(* PLC project Pizzarpocessor_03_11_2025.project, CODESYS CODESYS V3.5 SP21 Patch 1 *)
(* stored: creationDateTime 2025-11-18T11:47:58.0390156, modificationDateTime 2025-11-12T10:55:39.9225124 *)

TYPE HopperState : (OFF, IDLE, DISPENSING, LOW_LEVEL_FAULT, BLOCKED, MANUAL);
END_TYPE

TYPE ConveyorStatus : STRUCT
  Conveyor_ID : INT;  (* Conveyor number/ID *)
  Speed : REAL;  (* Percentage of speed *)
  Running : BOOL;
  State : ConveyorState;
  Ready : BOOL;  (* Interlock *)
END_STRUCT;
END_TYPE

TYPE HopperStatus : STRUCT
  Hopper_Id : INT;  (* Hopper Location/ID *)
  State : HopperState;  (* HopperState refering to ENUM *)
  Fill_Level : REAL;  (* Hopper_Ingredient level *)
  Ingredient_ID : INT;  (* Ingredient Name or Ingredient ID *)
  Alarm_Active : BOOL;  (* Alarm Status *)
  Ready : BOOL;  (* Interlock *)
  StartCount : DINT;
  LastFaultCode : INT;
  Timestamp : TIME;
END_STRUCT;
END_TYPE

TYPE ConveyorState : (OFF, IDLE, ON, JAM_FAULT, MANUAL);
END_TYPE

TYPE VFDStatus : STRUCT
  VFD_ID : STRING(20);  (* Identification *)
  State : VFDState;
  SpeedSetpoint_Percentage : REAL;  (* Speed *)
  Speed_Actual : REAL;
  Speedactual_Hz : REAL;
  IsRunning : BOOL;  (* Status *)
  IsAtSpeed : BOOL;
  Ready : BOOL;
  Alarm_Active : BOOL;  (* Alarms *)
  LastFault_Code : INT;
  Interlock_REason : STRING(50);
  StartCount : UDINT;  (* Counters *)
  RunTime_Hours : REAL;
  Current : REAL;  (* Hardware_DATA *)
  Torque_Percentage : REAL;
  Comm_OK : BOOL;  (* Comms *)
  Comms_Fault_Code : INT;
  TimeStamp : TIME;  (* TimeStamp *)
END_STRUCT;
END_TYPE

(* values of VFDState: Starting: Ramp-up Phase; Running: Normal operation; Stopping: Controlled deceleration; Stopped: VFD Stopped; Idle: VFD Powered but not running; Fault: VFD in Fault State; E_Stop: E-Stop Condition *)

TYPE VFDState : (Starting, Running, Stopping, Stopped, Idle, Fault, E_Stop);
END_TYPE

PROGRAM Supervisor_PRG
  VAR
    PID : PID;
  END_VAR

                    PID(KP:=1,SET_POINT:=1,ACTUAL:=1,TN:=1,TV:=1);
	
                  
END_PROGRAM

FUNCTION_BLOCK FB_Hopper
  VAR_INPUT
    StartDispense : BOOL;
    StopDispense : BOOL;
    ResetFault : BOOL;
    UpstreamReady : BOOL;
    DownstreamReady : BOOL;
    SimMode : BOOL;
  END_VAR
  VAR_OUTPUT
    Status : HopperStatus;
  END_VAR
  VAR
    Timer_LowLevel : TON;  (* timer for low level fault *)
  END_VAR

                    
// Main State Machine
CASE Status.State OF
	
    HopperState.OFF:
        IF UpstreamReady AND DownstreamReady THEN
            Status.State := HopperState.IDLE;
        END_IF

    HopperState.IDLE:
        Status.Ready := Status.Fill_Level > 10.0 AND NOT Status.Alarm_Active;
        IF StartDispense AND Status.Ready THEN
            Status.State := HopperState.DISPENSING;
            Status.StartCount := Status.StartCount + 1;
        END_IF
        IF Status.Fill_Level < 5.0 THEN
            Status.State := HopperState.LOW_LEVEL_FAULT;
        END_IF

    HopperState.DISPENSING:
        IF SimMode THEN
            Status.Fill_Level := Status.Fill_Level - 0.1; // simulate use
        END_IF
        IF StopDispense THEN
            Status.State := HopperState.IDLE;
        END_IF
        IF Status.Fill_Level < 5.0 THEN
            Status.State := HopperState.LOW_LEVEL_FAULT;
        END_IF

    HopperState.LOW_LEVEL_FAULT:
        Status.Alarm_Active := TRUE;
        Status.LastFaultCode := 101; // code for low level fault
        IF ResetFault AND Status.Fill_Level > 10.0 THEN
            Status.Alarm_Active := FALSE;
            Status.State := HopperState.IDLE;
        END_IF

    HopperState.BLOCKED:
        // implement other block conditions (e.g., jammed/fault inputs)
        IF ResetFault THEN
            Status.State := HopperState.IDLE;
        END_IF
    HopperState.MANUAL:    // In MANUAL, the operator can force DISPENSING or IDLE
        IF StartDispense THEN  
            Status.State := HopperState.DISPENSING;
        ELSIF StopDispense THEN
	          Status.State := HopperState.IDLE;
        END_IF

    // Interlock: even in manual, block if safety is lost
    IF NOT UpstreamReady OR NOT DownstreamReady THEN
        Status.State := HopperState.BLOCKED;
    END_IF

END_CASE

// Diagnostic update
Status.Timestamp := TIME(); // update time on every scan
                  
END_FUNCTION_BLOCK

FUNCTION_BLOCK FB_Conveyor
  VAR_INPUT
    Start : BOOL;
    Stop : BOOL;
    ResetFault : BOOL;
    UpstreamReady : BOOL;
    DownstreamReady : BOOL;
    SimMode : BOOL;
    Speed_Setpoint : REAL;  (* percentage in speed *)
  END_VAR
  VAR_OUTPUT
    Current_Speed : REAL;
    Status : ConveyorStatus;
  END_VAR

                    IF NOT UpstreamReady OR NOT DownstreamReady THEN
    Status.State := ConveyorState.JAM_FAULT;
ELSE
    CASE Status.State OF
        ConveyorState.OFF:
            Status.Running := FALSE;
            Current_Speed := 0.0;
            Status.Ready := FALSE;
            IF UpstreamReady AND DownstreamReady THEN
                Status.State := ConveyorState.IDLE;
            END_IF

        ConveyorState.IDLE:
            Status.Running := FALSE;
            Current_Speed := 0.0;
            Status.Ready := TRUE;
            IF Start THEN
                Status.State := ConveyorState.ON;
            END_IF

        ConveyorState.ON:
            Status.Running := TRUE;
            Current_Speed := Speed_Setpoint;
            Status.Speed := Speed_Setpoint;
            Status.Ready := TRUE;
            IF Stop THEN
                Status.State := ConveyorState.OFF;
            END_IF

        ConveyorState.JAM_FAULT:
            Status.Running := FALSE;
            Current_Speed := 0.0;
            Status.Ready := FALSE;
            IF ResetFault THEN
                Status.State := ConveyorState.IDLE;
            END_IF

        ConveyorState.MANUAL:
            IF Start THEN
                Status.State := ConveyorState.ON;
            ELSIF Stop THEN
                Status.State := ConveyorState.OFF;
            END_IF
    END_CASE
END_IF

                  
END_FUNCTION_BLOCK

FUNCTION_BLOCK FB_VFD
  VAR_INPUT
    SpeedSetpoint_Percent : REAL;  (* Speed setpoint (0-100%) *)
    DirectionForward : BOOL := TRUE;  (* TRUE=Forward, FALSE=Reverse *)
    LidClosed : BOOL := TRUE;  (* Door/Lid interlock (mixer) *)
    UpstreamReady : BOOL := TRUE;  (* Upstream equipment ready *)
    DownstreamReady : BOOL := TRUE;  (* Downstream equipment ready *)
    EmergencyStop : BOOL := FALSE;  (* E-stop signal *)
    SimMode : BOOL := FALSE;  (* Simulation (like Hopper's SimMode) *)
  END_VAR
  VAR_OUTPUT
    Status : VFDStatus;  (* Status (like Hopper.Status) *)
    OUT_Run : BOOL;  (* Run command *)
    OUT_Forward : BOOL;  (* Forward direction *)
    OUT_Reverse : BOOL;  (* Reverse direction *)
    OUT_SpeedReference : REAL;  (* Speed reference (0-100%) *)
    OUT_FaultReset : BOOL;  (* Fault reset pulse *)
  END_VAR
  VAR
    _CmdStart : BOOL;  (* Internal command flags (set by methods) *)
    _CmdStop : BOOL;
    _CmdReset : BOOL;
    MotorRatedHz : REAL := 60.0;  (* Motor rated frequency *)
    AccelTime_s : REAL := 10.0;  (* Accel time (seconds) *)
    DecelTime_s : REAL := 10.0;  (* Decel time (seconds) *)
    SpeedRamped_Hz : REAL;  (* Speed control *)
    RampRate_Hz_per_sec : REAL;
    Timer_Starting : TON;  (* Timers (like Hopper's Timer_LowLevel) *)
    Timer_Stopping : TON;
    Timer_AtSpeed : TON;
    Timer_FaultReset : TON;
    RuntimeAccum : REAL;  (* Runtime tracking *)
    FirstScan : BOOL := TRUE;  (* First scan *)
    ScanTime : TIME := TIME#100ms;
    Trig_Reset : R_TRIG;  (* Triggers *)
  END_VAR

                    
                  
END_FUNCTION_BLOCK

CONFIGURATION Device
  RESOURCE Application ON PLC
    TASK MainTask(INTERVAL := T#20ms, PRIORITY := 1);
    TASK DatasourcesTask(INTERVAL := T#50ms, PRIORITY := 31);
    PROGRAM Supervisor_PRG WITH MainTask : Supervisor_PRG;
    PROGRAM Datasources.Datasources_PRG WITH DatasourcesTask : Datasources.Datasources_PRG;
  END_RESOURCE
END_CONFIGURATION
